{attribute 'linkalways'} 
{attribute 'no_explicit_call' := 'This FB is a CLASS and must be accessed using methods or properties'}
{attribute 'enable_dynamic_creation'}
FUNCTION_BLOCK FINAL MOD_BYTE EXTENDS Node
VAR
	in1 : _BYTE(0);
	in2 : _BYTE(0);
	out : _BYTE(0);
END_VAR

METHOD PUBLIC Clone : I_Node
VAR
	pNode : POINTER TO MOD_BYTE;
END_VAR
pNode := __NEW(MOD_BYTE);
Clone := pNode^;
END_METHOD

METHOD FB_init : BOOL
VAR_INPUT
	bInitRetains : BOOL; // if TRUE, the retain variables are initialized (warm start / cold start)
	bInCopyCode : BOOL;  // if TRUE, the instance afterwards gets moved into the copy code (online change)
END_VAR
AddInput('in1',THIS^.in1);
AddInput('in2',THIS^.in2);
AddOutput('out', THIS^.out);
END_METHOD

METHOD PROTECTED OnExecute
VAR
END_VAR
out.Value := in1.Value MOD in2.Value;
END_METHOD

END_FUNCTION_BLOCK

(* stored: Version 1.1.0.1, ProductVersion 3.1.4024.15
   POU MOD_BYTE: Id {4ec84a7d-ed10-4ee5-b2bd-456e7174249e}, SpecialFunc None
   Folder Constructor: Id {47831d9c-c829-4695-b049-af46828c4408}
   Method Clone: Id {8dbdbce5-a7ea-4427-ab6a-c37be7e1f0a4}
   Method FB_init: Id {4d558ade-5456-4b28-a705-e41d16b005d3}
   Method OnExecute: Id {10080b26-9ee1-4480-afdf-36a8c375dea8} *)
